(* PLC project Untitled1, Beckhoff Automation GmbH TF6420 Database Server Query Analyser 1.0.0.0 *)
(* stored: creationDateTime 2016-05-30T12:36:50, modificationDateTime 2016-05-30T12:36:50 *)

TYPE ST_DB_PID : STRUCT
  id : DINT;
  timestamp : DT;
  symbolname : STRING(255);
  aktiv : BOOL;
  w : STRING(45);
  KP : STRING(45);
  I : STRING(45);
  D : STRING(45);
  Ta : STRING(45);
  Einschalttoleranz : STRING(45);
  Offset : STRING(45);
END_STRUCT;
END_TYPE
